// TIA Portal V16 export
// export: Created 2024-10-15T16:30:45.030602Z, ExportSetting WithDefaults, DisplayName Totally Integrated Automation Portal, DisplayVersion V16, DisplayName TIA Portal Version Control Interface, DisplayVersion V16, DisplayName TIA Portal Openness, DisplayVersion V16, DisplayName STEP 7 Professional, DisplayVersion V16, DisplayName STEP 7 Safety, DisplayVersion V16, DisplayName WinCC Advanced, DisplayVersion V16
DATA_BLOCK "StanowiskoCiecia_1_DB"   // DB3
VERSION : 0.1
// stored: AutoNumber true, InstanceOfName StanowiskoCiecia, InstanceOfType FB
"StanowiskoCiecia"
   // VAR_INPUT
   //    iLiczbaCiecZadana : Int;
   //    xSygnalWyzwalajacy : Bool;
   //    xResetLicznika : Bool;
   // END_VAR
   // VAR_OUTPUT
   //    xZlecenieWToku : Bool;
   //    xZlecenieZakonczone : Bool;
   // END_VAR
   // VAR_IN_OUT
   //    iLicznikCiec : Int;
   // END_VAR
   // VAR
   //    xBitPamieci : Bool;
   // END_VAR
BEGIN
END_DATA_BLOCK
